{attribute addProperty BoxType "EJ7211-0010-0026"}
{attribute addProperty Id "ControlwordAT %Q*UINT162"}
{attribute addProperty CRC "1098258280"}
{attribute addProperty SizeInBites "16"}
{attribute addProperty SizeInBytes "2"}
TYPE DRV_Controlword_41761768 :
STRUCT
	{attribute addProperty Name "Controlword"}
	Controlword AT %Q* : UINT;
END_STRUCT
END_TYPE

(* stored: Version 1.2.0.0, ProductVersion 3.1.4024.9
   DUT DRV_Controlword_41761768: Id {4751bcbf-8a75-4954-8a03-a3ef8557fcd7} *)
